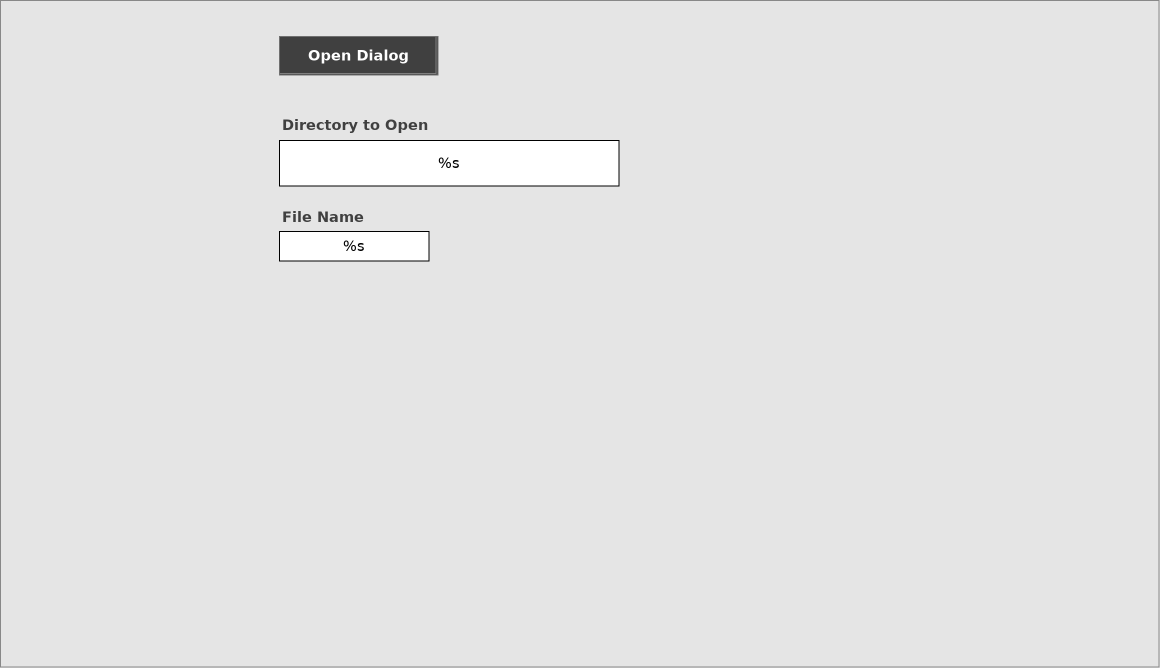
VISUALIZATION V_FileDialog  // 1160x668
    Button (279,36 159x39), "Open Dialog"
        tap P_FileDialog.bOpen
        OnMouseDown: OpenDialog Dialog=VisuDialogs.FileOpenSave, Parameters={fileListProvider: P_FileDialog.fbFileList}, OpenModal=True, OpenCentered=True
    Rectangle (279,231 150x30), "%s", text variable: P_FileDialog.sSelectedFileName
    Textfield (279,140 340x46), "%s", text variable: P_FileDialog.sDir
        OnMouseClick: write the text variable via Edit
    Label (279,107 264x36), "Directory to Open"
    Label (279,199 264x36), "File Name"
END_VISUALIZATION

(* stored: Version 1.1.0.1, ProductVersion 3.1.4024.3
   Visu V_FileDialog: Id {76aa7add-a667-429b-aa25-a76529f02c51} *)
